{attribute 'TcGenerated'}
{attribute 'no-analysis'}
{attribute 'linkalways'}
// This function has been automatically generated from the project information.
VAR_GLOBAL CONSTANT
	{attribute 'const_non_replaced'}
	stLibVersion_TwinCAT_Hashing_Algorithms : ST_LibVersion := (iMajor := 0, iMinor := 1, iBuild := 0, iRevision := 0, nFlags := 0, sVersion := '0.1.0.0');
END_VAR

(* stored: Version 1.1.0.1, ProductVersion 3.1.4024.4
   GVL Global_Version: Id {0e11180c-f160-42d3-b201-cf0ed22ab993} *)
